TYPE E_ModeRGB :
(
	eModeRGB_Off,
	eModeRGB_MANUAL,
	eModeRGB_AUTO,
	eModeRGB_AUTOREVERS
);
END_TYPE

(* stored: Version 1.1.0.1, ProductVersion 3.1.4018.5
   DUT E_ModeRGB: Id {c75de3a8-a58f-4695-81c0-44142652c1df} *)
